(* CODESYS project 3dom.project
   Title: 3dom
   Author: keny
   Version: 0.0.0.14

Project tree, tasks and I/O mapping:
  MyController : TM241CE40T/U, Schneider Electric, order no. TM241CE40T/U, version 4.0.6.18
    application Application
      libraries: Toolbox_Advance, 1.0.1.0 (Schneider Electric); Toolbox, 2.2.0.0 (Schneider Electric)
      task MAST (cyclic, interval 20 ms, priority 15, watchdog 100 ms x 1) calls Program_1
      task VISU_TASK (cyclic, interval 100 ms, priority 30) calls VisuElems.Visu_Prg
      global variables GVL
      visualisation Visualization
      visualisation Visualization_1
    DI : Digital Inputs, Schneider Electric, version 4.0.6.18
        input  M1 : DWORD  // IDW0
        input  lampa_1_kuchania_1_1_wl : BOOL  // IDW0.I0
        input  led_1_kuchnia_1_1_wl : BOOL  // IDW0.I1
        input  kinkiet_1_jadalnia_1_1_wl : BOOL  // IDW0.I2
        input  kinkiet_1_salon_1_1_wl : BOOL  // IDW0.I3
        input  kinkiet_2_salon_1_1_wl : BOOL  // IDW0.I4
        input  kinkiet_3_salon_1_1_wl : BOOL  // IDW0.I5
        input  led_1_salon_1_1_wl : BOOL  // IDW0.I6
        input  lampa_1_salon_1_1_wl : BOOL  // IDW0.I7
        input  lampa_1_jadalnia_1_1_wl : BOOL  // IDW0.I8
        input  kinkiet_1_schody_1_1_wl : BOOL  // IDW0.I9
        input  lampa_zew_wej_1_1_wl : BOOL  // IDW0.I10
        input  lampa_1_przedsionek_1_1_wl : BOOL  // IDW0.I11
        input  lampa_1_korytarz_1_1_wl : BOOL  // IDW0.I12
        input  lampa_1_pokoj_1_1_wl : BOOL  // IDW0.I13
        input  lampa_1_pokoj_2_1_wl : BOOL  // IDW0.I14
        input  kinkiet_1_pokoj_2_1_wl : BOOL  // IDW0.I15
        input  lampa_2_korytarz_1_1_wl : BOOL  // IDW0.I16
        input  lampa_pom_tech_1_1_wl : BOOL  // IDW0.I17
        input  lampa_1_lazienka_1_1_wl : BOOL  // IDW0.I18
        input  kinkiet_1_lazienka_1_1_wl : BOOL  // IDW0.I19
        input  lampa_zew_1_1_wl : BOOL  // IDW0.I20
        input  lampa_zew_2_1_wl : BOOL  // IDW0.I21
        input  lampa_zew_3_1_wl : BOOL  // IDW0.I22
        input  lampa_zew_4_1_wl : BOOL  // IDW0.I23
        input  ibDI_IB1 : BYTE  // IB1
    DQ : Digital Outputs, Schneider Electric, version 4.0.6.18
        output lampa_1_kuchania_1_1_rel : BOOL  // QW0.Q0
        output led_1_kuchnia_1_1_rel : BOOL  // QW0.Q1
        output kinkiet_1_jadalnia_1_1_rel : BOOL  // QW0.Q2
        output kinkiet_1_salon_1_1_rel : BOOL  // QW0.Q3
        output kinkiet_2_salon_1_1_rel : BOOL  // QW0.Q4
        output kinkiet_3_salon_1_1_rel : BOOL  // QW0.Q5
        output led_1_salon_1_1_rel : BOOL  // QW0.Q6
        output lampa_1_salon_1_1_rel : BOOL  // QW0.Q7
        output lampa_1_jadalnia_1_1_rel : BOOL  // QW0.Q8
        output kinkiet_1_schody_1_1_rel : BOOL  // QW0.Q9
        output lampa_zew_wej_1_1_rel : BOOL  // QW0.Q10
        output lampa_1_przedsionek_1_1_rel : BOOL  // QW0.Q11
        output lampa_1_korytarz_1_1_rel : BOOL  // QW0.Q12
        output lampa_1_pokoj_1_1_rel : BOOL  // QW0.Q13
        output lampa_1_pokoj_2_1_rel : BOOL  // QW0.Q14
        output kinkiet_1_pokoj_2_1_rel : BOOL  // QW0.Q15
        unmapped channels: QW0, QB1
    Counters : Counters, Schneider Electric, version 4.0.6.18
    Pulse_Generators : Pulse Generators, Schneider Electric, version 4.0.6.18
    Cartridge_1 : Cartridge, Schneider Electric, version 4.0.6.18
    Cartridge_2 : Cartridge, Schneider Electric, version 4.0.6.18
    IO_Bus : IO bus - TM3, Schneider Electric, version 4.0.6.18
      M2 : TM3DI16/G, Schneider Electric, order no. TM3DI16/G, version 1.0.1.4
          input  M2 : WORD  // IW0
          input  lampa_1_pokoj_3_1_wl : BOOL  // IW0.I0
          input  lampa_1_pom_gosp_1_1_wl : BOOL  // IW0.I1
          input  lampa_1_pokoj_4_1_wl : BOOL  // IW0.I2
          input  lampa_2_pokoj_4_1_wl : BOOL  // IW0.I3
          input  lampa_1_pokoj_5_1_wl : BOOL  // IW0.I4
          input  kinkiet_1_pokoj_5_1_wl : BOOL  // IW0.I5
          input  lampa_1_korytarz_2_1_wl : BOOL  // IW0.I6
          input  led_1_korytarz_2_1_wl : BOOL  // IW0.I7
          input  lampa_1_lazienka_2_1_wl : BOOL  // IW0.I8
          input  kinkiet_1_lazienka_2_1_wl : BOOL  // IW0.I9
          input  kinkiet_2_lazienka_2_1_wl : BOOL  // IW0.I10
          input  lampa_1_pralnia_1_1_wl : BOOL  // IW0.I11
          input  lampa_1_garderoba_1_1_wl : BOOL  // IW0.I12
          input  os_ogrodu_1_1_wl : BOOL  // IW0.I13
          input  kinkiet_4_salon_1_1_wl : BOOL  // IW0.I14
          input  kinkiet_2_schody_1_1_wl : BOOL  // IW0.I15
      M5 : TM3DQ16T/G, Schneider Electric, order no. TM3DQ16T/G, version 1.0.1.4
          output lampa_1_lazienka_2_1_rel : BOOL  // QB0.Q0
          output kinkiet_1_lazienka_2_1_rel : BOOL  // QB0.Q1
          output kinkiet_2_lazienka_2_1_rel : BOOL  // QB0.Q2
          output lampa_1_pralnia_1_1_rel : BOOL  // QB0.Q3
          output lampa_1_garderoba_1_1_rel : BOOL  // QB0.Q4
          output os_ogrodu_1_1_rel : BOOL  // QB0.Q5
          output kinkiet_4_salon_1_1_rel : BOOL  // QB0.Q6
          output kinkiet_2_schody_1_1_rel : BOOL  // QB0.Q7
          output lampa_zew_5_1_rel : BOOL  // QB0.Q8
          unmapped channels: QB0
      M3 : TM3DI16/G, Schneider Electric, order no. TM3DI16/G, version 1.0.1.4
          input  M3 : WORD  // IW0
          input  lampa_zew_5_1_wl : BOOL  // IW0.I0
          input  wlacz_lampy : BOOL  // IW0.I1
          input  wylacz_lampy : BOOL  // IW0.I2
      M4 : TM3DQ16T/G, Schneider Electric, order no. TM3DQ16T/G, version 1.0.1.4
          output lampa_2_korytarz_1_1_rel : BOOL  // QB0.Q0
          output lampa_pom_tech_1_1_rel : BOOL  // QB0.Q1
          output lampa_1_lazienka_1_1_rel : BOOL  // QB0.Q2
          output kinkiet_1_lazienka_1_1_rel : BOOL  // QB0.Q3
          output lampa_zew_1_1_rel : BOOL  // QB0.Q4
          output lampa_zew_2_1_rel : BOOL  // QB0.Q5
          output lampa_zew_3_1_rel : BOOL  // QB0.Q6
          output lampa_zew_4_1_rel : BOOL  // QB0.Q7
          output lampa_1_pokoj_3_1_rel : BOOL  // QB0.Q8
          output lampa_1_pom_gosp_1_1_rel : BOOL  // QB0.Q9
          output lampa_1_pokoj_4_1_rel : BOOL  // QB0.Q10
          output lampa_2_pokoj_4_1_rel : BOOL  // QB0.Q11
          output lampa_1_pokoj_5_1_rel : BOOL  // QB0.Q12
          output kinkiet_1_pokoj_5_1_rel : BOOL  // QB0.Q13
          output lampa_1_korytarz_2_1_rel : BOOL  // QB0.Q14
          output led_1_korytarz_2_1_rel : BOOL  // QB0.Q15
          unmapped channels: QB0
      M6 : TM3DQ16R/G, Schneider Electric, order no. TM3DQ16R/G, version 1.0.1.4
          output zawor_woda_ogrod_1_rel : BOOL  // QW0.Q0
          output ogrzewanie_zawor_1_1_rel : BOOL  // QW0.Q1
          output ogrzewanie_zawor_2_1_rel : BOOL  // QW0.Q2
          output ogrzewanie_zawor_3_1_rel : BOOL  // QW0.Q3
          output ogrzewanie_zawor_4_1_rel : BOOL  // QW0.Q4
          output ogrzewanie_zawor_5_1_rel : BOOL  // QW0.Q5
          output ogrzewanie_zawor_6_1_rel : BOOL  // QW0.Q6
          output ogrzewanie_zawor_7_1_rel : BOOL  // QW0.Q7
          output ogrzewanie_zawor_8_1_rel : BOOL  // QW0.Q8
          unmapped channels: QW0
    COM_Bus : COM bus, Schneider Electric, version 4.0.6.18
    Ethernet_1 : Ethernet Network, Schneider Electric, version 4.0.6.18
        settings: DeviceName = 'nodeZ'; WebServer = TRUE; FTP Server = TRUE; SoMachine Protocol = TRUE; Modbus Server = TRUE; NetManage Protocol = TRUE; SNMP protocol = TRUE; Enable Routing = FALSE; WebVisu protocol = TRUE; DHCP Server Active = TRUE
    Serial_Line_1 : Serial line, Schneider Electric, version 4.0.6.18
      SoMachine_Network_Manager : SoMachine-Network Manager, Schneider Electric, version 4.0.0.2
    Serial_Line_2 : Serial line, Schneider Electric, version 4.0.6.18
      Modbus_Manager : Modbus Manager, Schneider Electric, version 4.0.0.2
  libraries: Standard, * (System)
  function block swichOnOffFUNC [LD]
  function block lightFUNC [LD]
  program Program_1 [LD]
  text list GlobalTextList
  GlobalImagePool
  5ce3da45-db07-42e7-a21c-a00fff4ed8f6|parter.JPG
*)

// MyController/Application/GVL
VAR_GLOBAL 
	;
END_VAR

// Program_1
PROGRAM Program_1
VAR
	lampa_1_kuchania_1_1_DB: swichOnOffFUNC;
	kinkiet_1_jadalnia_1_1_DB: swichOnOffFUNC;
	led_1_kuchnia_1_1_DB: swichOnOffFUNC;
	kinkiet_1_salon_1_1_DB: swichOnOffFUNC;
	kinkiet_2_salon_1_1_DB: swichOnOffFUNC;
	kinkiet_3_salon_1_1_DB: swichOnOffFUNC;
	led_1_salon_1_1_DB: swichOnOffFUNC;
	lampa_1_salon_1_1_DB: swichOnOffFUNC;
	lampa_1_jadalnia_1_1_DB: swichOnOffFUNC;
	kinkiet_1_schody_1_1_DB: swichOnOffFUNC;
	lampa_1_zew_wejsc_1_1_DB: swichOnOffFUNC;
	lampa_1_przedsionek_1_1_DB: swichOnOffFUNC;
	lampa_1_korytarz_1_1_db: swichOnOffFUNC;
	lampa_1_pokoj_1_1_wl_DB: swichOnOffFUNC;
	lampa_1_pokoj_2_1_DB: swichOnOffFUNC;
	kinkiet_1_pokoj_2_1_DB: swichOnOffFUNC;
	lampa_1_korytarz_1_2_DB: swichOnOffFUNC;
	lampa_1_pokoj_1_1_DB: swichOnOffFUNC;
	lampa_2_korytarz_1_1_DB: swichOnOffFUNC;
	lampa_pom_tech_1_1_DB: swichOnOffFUNC;
	lampa_1_laz_1_1_DB: swichOnOffFUNC;
	lampa_1_lazienka_1_1_DB: swichOnOffFUNC;
	kinkiet_1_lazienka_1_1_DB: swichOnOffFUNC;
	lampa_zew_1_1_DB: swichOnOffFUNC;
	lampa_zew_2_1_DB: swichOnOffFUNC;
	lampa_zew_3_1_DB: swichOnOffFUNC;
	lampa_zew_4_1_DB: swichOnOffFUNC;
	lampa_1_pokoj_3_1_DB: swichOnOffFUNC;
	lampa_1_pom_gosp_1_1_DB: swichOnOffFUNC;
	lampa_1_pokoj_4_1_DB: swichOnOffFUNC;
	lampa_2_pokoj_4_1_DB: swichOnOffFUNC;
	lampa_1_pokoj_5_1_DB: swichOnOffFUNC;
	kinkiet_1_pokoj_5_1_DB: swichOnOffFUNC;
	lampa_1_korytarz_2_1_DB: swichOnOffFUNC;
	led_1_korytarz_2_1_DB: swichOnOffFUNC;
	lampa_1_lazienka_2_1_DB: swichOnOffFUNC;
	kinkiet_1_lazienka_2_1_DB: swichOnOffFUNC;
	kinkiet_2_lazienka_2_1_DB: swichOnOffFUNC;
	lampa_1_pralnia_1_1_DB: swichOnOffFUNC;
	lampa_1_garderoba_1_1_DB: swichOnOffFUNC;
	os_ogrodu_1_1_DB: swichOnOffFUNC;
	kinkiet_4_salon_1_1_DB: swichOnOffFUNC;
	kinkiet_2_schody_1_1_DB: swichOnOffFUNC;
	lampa_zew_5_1_DB: swichOnOffFUNC;
	wlacz_lampy_DB: swichOnOffFUNC;
	lamp_zewnetrzna_1: BOOL;
	lampa_zewnetrzna_5_visu: BOOL;
	lampa_1_kuchania_visu: BOOL;
	led_1_kuchnia_1_1_visu: BOOL;
	kinkiet_1_jadalnia_1_1_visu: BOOL;
	kinkiet_1_salon_1_1_visu: BOOL;
	kinkiet_2_salon_1_1_visu: BOOL;
	kinkiet_3_salon_1_1_visu: BOOL;
	lampa_1_salon_1_1_visu: BOOL;
	lampa_1_jadalnia_1_1_visu: BOOL;
	kinkiet_1_schody_1_1_visu: BOOL;
	lampa_zew_wej_1_1_visu: BOOL;
	lampa_1_przedsionek_1_1_visu: BOOL;
	lampa_1_korytarz_1_1_visu: BOOL;
	lampa_1_pokoj_1_1_visu: BOOL;
	lampa_1_pokoj_2_1_visu: BOOL;
	led_1_kuchnia_visu: BOOL;
	lampa_2_korytarz_1_1_VISU: BOOL;
	kinkiet_1_pokoj_2_1_visu: BOOL;
	lampa_pom_tech_1_1_visu: BOOL;
	lampa_1_lazienka_1_1_visu: BOOL;
	kinkiet_1_lazienka_1_1_visu: BOOL;
	lampa_zew_1_1_visu: BOOL;
	lampa_zew_2_1_visu: BOOL;
	lampa_zew_3_1_visu: BOOL;
	lampa_zew_4_1_visu: BOOL;
	lampa_1_pokoj_3_1_visu: BOOL;
	lampa_1_pom_gosp_1_1_visu: BOOL;
	lampa_1_pokoj_4_1_visu: BOOL;
	lampa_2_pokoj_4_1_visu: BOOL;
	lampa_1_pokoj_5_1_visu: BOOL;
	kinkiet_1_pokoj_5_1_visu: BOOL;
	lampa_1_korytarz_2_1_visu: BOOL;
	led_1_korytarz_2_1_visu: BOOL;
	lampa_1_lazienka_2_1_visu: BOOL;
	kinkiet_1_lazienka_2_1_visu: BOOL;
	kinkiet_2_lazienka_2_1_visu: BOOL;
	lampa_1_pralnia_1_1_visu: BOOL;
	lampa_1_garderoba_1_1_visu: BOOL;
	os_ogrodu_1_1_visu: BOOL;
	kinkiet_4_salon_1_1_visu: BOOL;
	kinkiet_2_schody_1_1_visu: BOOL;
	lampa_zew_5_1_visu: BOOL;
	led_1_salon_1_1_visu: BOOL;
END_VAR

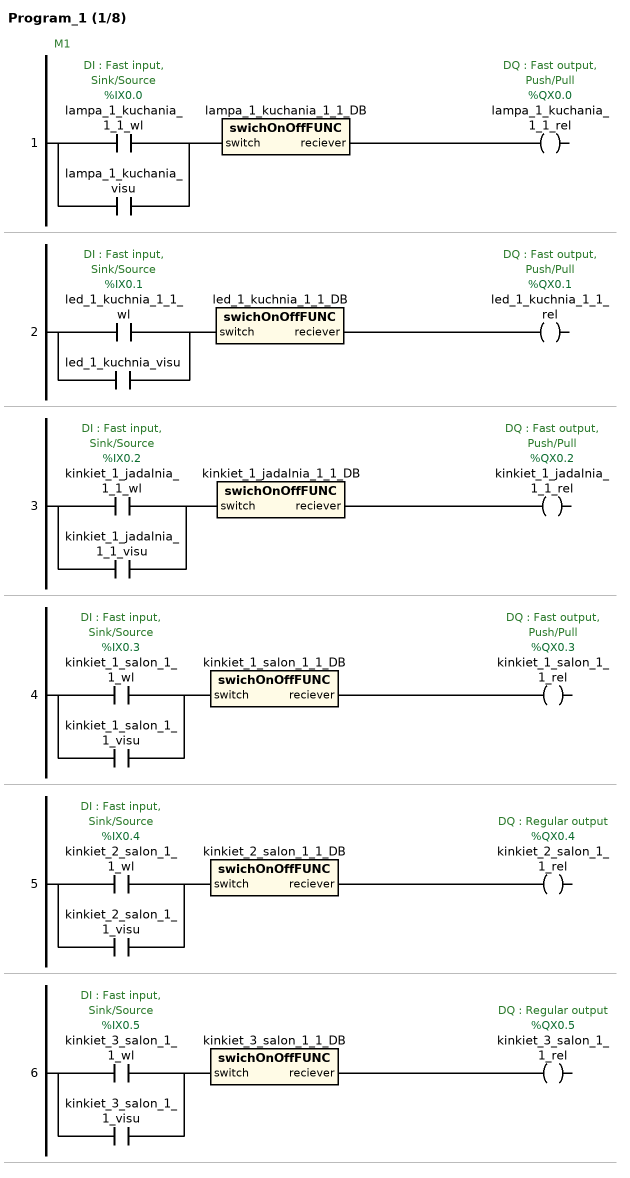
// NETWORK 1
// M1
//   lampa_1_kuchania_1_1_wl: DI : Fast input, Sink/Source | AT %IX0.0
//   lampa_1_kuchania_1_1_rel: DQ : Fast output, Push/Pull | AT %QX0.0
lampa_1_kuchania_1_1_DB(switch := lampa_1_kuchania_1_1_wl OR lampa_1_kuchania_visu); // swichOnOffFUNC
lampa_1_kuchania_1_1_rel := lampa_1_kuchania_1_1_DB.reciever;

// NETWORK 2
//   led_1_kuchnia_1_1_wl: DI : Fast input, Sink/Source | AT %IX0.1
//   led_1_kuchnia_1_1_rel: DQ : Fast output, Push/Pull | AT %QX0.1
led_1_kuchnia_1_1_DB(switch := led_1_kuchnia_1_1_wl OR led_1_kuchnia_visu); // swichOnOffFUNC
led_1_kuchnia_1_1_rel := led_1_kuchnia_1_1_DB.reciever;

// NETWORK 3
//   kinkiet_1_jadalnia_1_1_wl: DI : Fast input, Sink/Source | AT %IX0.2
//   kinkiet_1_jadalnia_1_1_rel: DQ : Fast output, Push/Pull | AT %QX0.2
kinkiet_1_jadalnia_1_1_DB(switch := kinkiet_1_jadalnia_1_1_wl OR kinkiet_1_jadalnia_1_1_visu); // swichOnOffFUNC
kinkiet_1_jadalnia_1_1_rel := kinkiet_1_jadalnia_1_1_DB.reciever;

// NETWORK 4
//   kinkiet_1_salon_1_1_wl: DI : Fast input, Sink/Source | AT %IX0.3
//   kinkiet_1_salon_1_1_rel: DQ : Fast output, Push/Pull | AT %QX0.3
kinkiet_1_salon_1_1_DB(switch := kinkiet_1_salon_1_1_wl OR kinkiet_1_salon_1_1_visu); // swichOnOffFUNC
kinkiet_1_salon_1_1_rel := kinkiet_1_salon_1_1_DB.reciever;

// NETWORK 5
//   kinkiet_2_salon_1_1_wl: DI : Fast input, Sink/Source | AT %IX0.4
//   kinkiet_2_salon_1_1_rel: DQ : Regular output | AT %QX0.4
kinkiet_2_salon_1_1_DB(switch := kinkiet_2_salon_1_1_wl OR kinkiet_2_salon_1_1_visu); // swichOnOffFUNC
kinkiet_2_salon_1_1_rel := kinkiet_2_salon_1_1_DB.reciever;

// NETWORK 6
//   kinkiet_3_salon_1_1_wl: DI : Fast input, Sink/Source | AT %IX0.5
//   kinkiet_3_salon_1_1_rel: DQ : Regular output | AT %QX0.5
kinkiet_3_salon_1_1_DB(switch := kinkiet_3_salon_1_1_wl OR kinkiet_3_salon_1_1_visu); // swichOnOffFUNC
kinkiet_3_salon_1_1_rel := kinkiet_3_salon_1_1_DB.reciever;

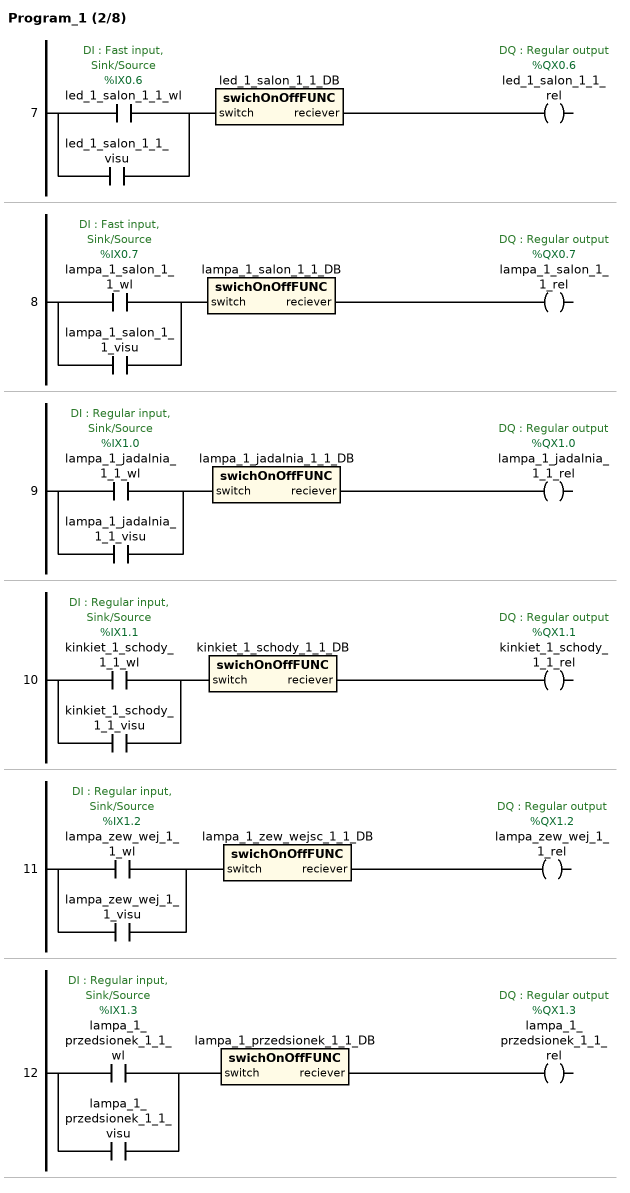
// NETWORK 7
//   led_1_salon_1_1_wl: DI : Fast input, Sink/Source | AT %IX0.6
//   led_1_salon_1_1_rel: DQ : Regular output | AT %QX0.6
led_1_salon_1_1_DB(switch := led_1_salon_1_1_wl OR led_1_salon_1_1_visu); // swichOnOffFUNC
led_1_salon_1_1_rel := led_1_salon_1_1_DB.reciever;

// NETWORK 8
//   lampa_1_salon_1_1_wl: DI : Fast input, Sink/Source | AT %IX0.7
//   lampa_1_salon_1_1_rel: DQ : Regular output | AT %QX0.7
lampa_1_salon_1_1_DB(switch := lampa_1_salon_1_1_wl OR lampa_1_salon_1_1_visu); // swichOnOffFUNC
lampa_1_salon_1_1_rel := lampa_1_salon_1_1_DB.reciever;

// NETWORK 9
//   lampa_1_jadalnia_1_1_wl: DI : Regular input, Sink/Source | AT %IX1.0
//   lampa_1_jadalnia_1_1_rel: DQ : Regular output | AT %QX1.0
lampa_1_jadalnia_1_1_DB(switch := lampa_1_jadalnia_1_1_wl OR lampa_1_jadalnia_1_1_visu); // swichOnOffFUNC
lampa_1_jadalnia_1_1_rel := lampa_1_jadalnia_1_1_DB.reciever;

// NETWORK 10
//   kinkiet_1_schody_1_1_wl: DI : Regular input, Sink/Source | AT %IX1.1
//   kinkiet_1_schody_1_1_rel: DQ : Regular output | AT %QX1.1
kinkiet_1_schody_1_1_DB(switch := kinkiet_1_schody_1_1_wl OR kinkiet_1_schody_1_1_visu); // swichOnOffFUNC
kinkiet_1_schody_1_1_rel := kinkiet_1_schody_1_1_DB.reciever;

// NETWORK 11
//   lampa_zew_wej_1_1_wl: DI : Regular input, Sink/Source | AT %IX1.2
//   lampa_zew_wej_1_1_rel: DQ : Regular output | AT %QX1.2
lampa_1_zew_wejsc_1_1_DB(switch := lampa_zew_wej_1_1_wl OR lampa_zew_wej_1_1_visu); // swichOnOffFUNC
lampa_zew_wej_1_1_rel := lampa_1_zew_wejsc_1_1_DB.reciever;

// NETWORK 12
//   lampa_1_przedsionek_1_1_wl: DI : Regular input, Sink/Source | AT %IX1.3
//   lampa_1_przedsionek_1_1_rel: DQ : Regular output | AT %QX1.3
lampa_1_przedsionek_1_1_DB(switch := lampa_1_przedsionek_1_1_wl OR lampa_1_przedsionek_1_1_visu); // swichOnOffFUNC
lampa_1_przedsionek_1_1_rel := lampa_1_przedsionek_1_1_DB.reciever;

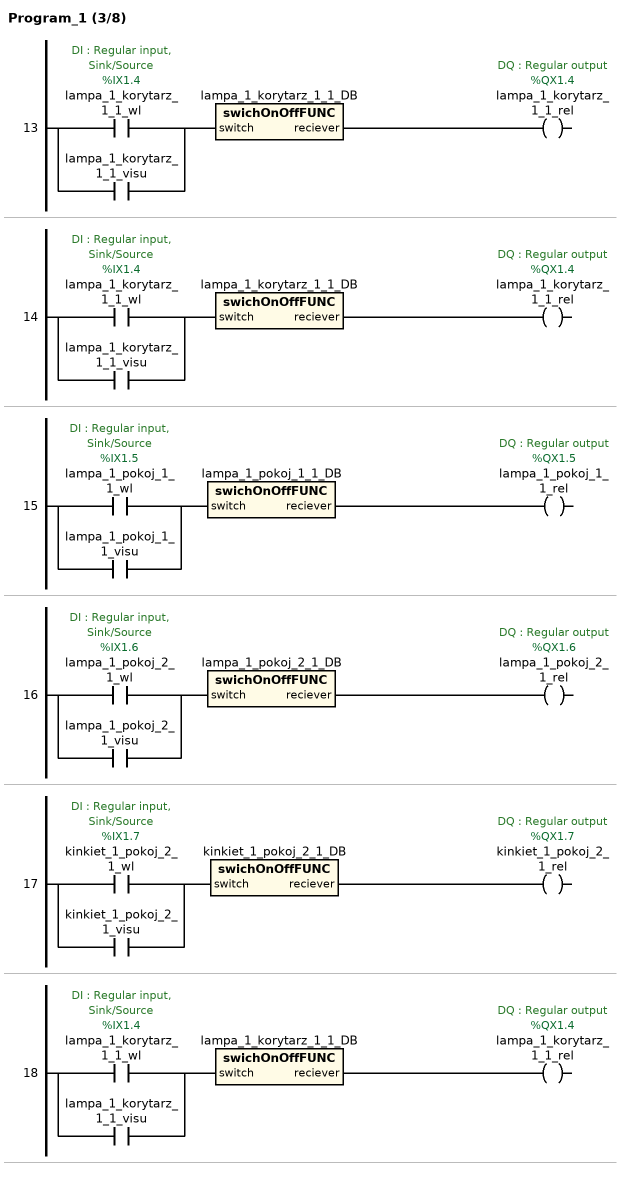
// NETWORK 13
//   lampa_1_korytarz_1_1_wl: DI : Regular input, Sink/Source | AT %IX1.4
//   lampa_1_korytarz_1_1_rel: DQ : Regular output | AT %QX1.4
lampa_1_korytarz_1_1_DB(switch := lampa_1_korytarz_1_1_wl OR lampa_1_korytarz_1_1_visu); // swichOnOffFUNC
lampa_1_korytarz_1_1_rel := lampa_1_korytarz_1_1_DB.reciever;

// NETWORK 14
//   lampa_1_korytarz_1_1_wl: DI : Regular input, Sink/Source | AT %IX1.4
//   lampa_1_korytarz_1_1_rel: DQ : Regular output | AT %QX1.4
lampa_1_korytarz_1_1_DB(switch := lampa_1_korytarz_1_1_wl OR lampa_1_korytarz_1_1_visu); // swichOnOffFUNC
lampa_1_korytarz_1_1_rel := lampa_1_korytarz_1_1_DB.reciever;

// NETWORK 15
//   lampa_1_pokoj_1_1_wl: DI : Regular input, Sink/Source | AT %IX1.5
//   lampa_1_pokoj_1_1_rel: DQ : Regular output | AT %QX1.5
lampa_1_pokoj_1_1_DB(switch := lampa_1_pokoj_1_1_wl OR lampa_1_pokoj_1_1_visu); // swichOnOffFUNC
lampa_1_pokoj_1_1_rel := lampa_1_pokoj_1_1_DB.reciever;

// NETWORK 16
//   lampa_1_pokoj_2_1_wl: DI : Regular input, Sink/Source | AT %IX1.6
//   lampa_1_pokoj_2_1_rel: DQ : Regular output | AT %QX1.6
lampa_1_pokoj_2_1_DB(switch := lampa_1_pokoj_2_1_wl OR lampa_1_pokoj_2_1_visu); // swichOnOffFUNC
lampa_1_pokoj_2_1_rel := lampa_1_pokoj_2_1_DB.reciever;

// NETWORK 17
//   kinkiet_1_pokoj_2_1_wl: DI : Regular input, Sink/Source | AT %IX1.7
//   kinkiet_1_pokoj_2_1_rel: DQ : Regular output | AT %QX1.7
kinkiet_1_pokoj_2_1_DB(switch := kinkiet_1_pokoj_2_1_wl OR kinkiet_1_pokoj_2_1_visu); // swichOnOffFUNC
kinkiet_1_pokoj_2_1_rel := kinkiet_1_pokoj_2_1_DB.reciever;

// NETWORK 18
//   lampa_1_korytarz_1_1_wl: DI : Regular input, Sink/Source | AT %IX1.4
//   lampa_1_korytarz_1_1_rel: DQ : Regular output | AT %QX1.4
lampa_1_korytarz_1_1_DB(switch := lampa_1_korytarz_1_1_wl OR lampa_1_korytarz_1_1_visu); // swichOnOffFUNC
lampa_1_korytarz_1_1_rel := lampa_1_korytarz_1_1_DB.reciever;

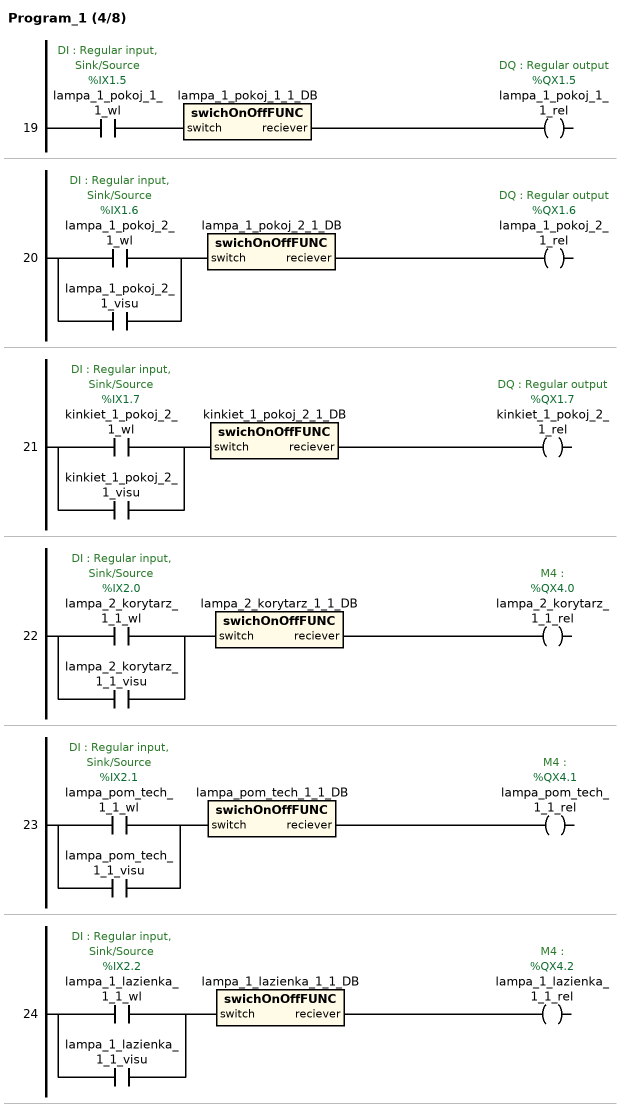
// NETWORK 19
//   lampa_1_pokoj_1_1_wl: DI : Regular input, Sink/Source | AT %IX1.5
//   lampa_1_pokoj_1_1_rel: DQ : Regular output | AT %QX1.5
lampa_1_pokoj_1_1_DB(switch := lampa_1_pokoj_1_1_wl); // swichOnOffFUNC
lampa_1_pokoj_1_1_rel := lampa_1_pokoj_1_1_DB.reciever;

// NETWORK 20
//   lampa_1_pokoj_2_1_wl: DI : Regular input, Sink/Source | AT %IX1.6
//   lampa_1_pokoj_2_1_rel: DQ : Regular output | AT %QX1.6
lampa_1_pokoj_2_1_DB(switch := lampa_1_pokoj_2_1_wl OR lampa_1_pokoj_2_1_visu); // swichOnOffFUNC
lampa_1_pokoj_2_1_rel := lampa_1_pokoj_2_1_DB.reciever;

// NETWORK 21
//   kinkiet_1_pokoj_2_1_wl: DI : Regular input, Sink/Source | AT %IX1.7
//   kinkiet_1_pokoj_2_1_rel: DQ : Regular output | AT %QX1.7
kinkiet_1_pokoj_2_1_DB(switch := kinkiet_1_pokoj_2_1_wl OR kinkiet_1_pokoj_2_1_visu); // swichOnOffFUNC
kinkiet_1_pokoj_2_1_rel := kinkiet_1_pokoj_2_1_DB.reciever;

// NETWORK 22
//   lampa_2_korytarz_1_1_wl: DI : Regular input, Sink/Source | AT %IX2.0
//   lampa_2_korytarz_1_1_rel: M4 : | AT %QX4.0
lampa_2_korytarz_1_1_DB(switch := lampa_2_korytarz_1_1_wl OR lampa_2_korytarz_1_1_visu); // swichOnOffFUNC
lampa_2_korytarz_1_1_rel := lampa_2_korytarz_1_1_DB.reciever;

// NETWORK 23
//   lampa_pom_tech_1_1_wl: DI : Regular input, Sink/Source | AT %IX2.1
//   lampa_pom_tech_1_1_rel: M4 : | AT %QX4.1
lampa_pom_tech_1_1_DB(switch := lampa_pom_tech_1_1_wl OR lampa_pom_tech_1_1_visu); // swichOnOffFUNC
lampa_pom_tech_1_1_rel := lampa_pom_tech_1_1_DB.reciever;

// NETWORK 24
//   lampa_1_lazienka_1_1_wl: DI : Regular input, Sink/Source | AT %IX2.2
//   lampa_1_lazienka_1_1_rel: M4 : | AT %QX4.2
lampa_1_lazienka_1_1_DB(switch := lampa_1_lazienka_1_1_wl OR lampa_1_lazienka_1_1_visu); // swichOnOffFUNC
lampa_1_lazienka_1_1_rel := lampa_1_lazienka_1_1_DB.reciever;

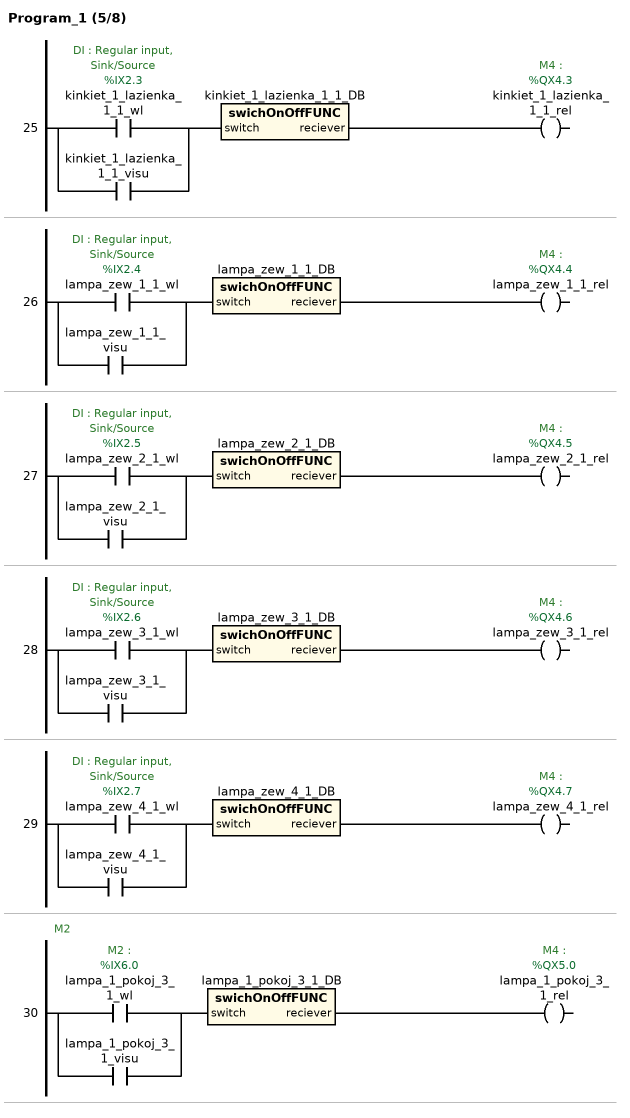
// NETWORK 25
//   kinkiet_1_lazienka_1_1_wl: DI : Regular input, Sink/Source | AT %IX2.3
//   kinkiet_1_lazienka_1_1_rel: M4 : | AT %QX4.3
kinkiet_1_lazienka_1_1_DB(switch := kinkiet_1_lazienka_1_1_wl OR kinkiet_1_lazienka_1_1_visu); // swichOnOffFUNC
kinkiet_1_lazienka_1_1_rel := kinkiet_1_lazienka_1_1_DB.reciever;

// NETWORK 26
//   lampa_zew_1_1_wl: DI : Regular input, Sink/Source | AT %IX2.4
//   lampa_zew_1_1_rel: M4 : | AT %QX4.4
lampa_zew_1_1_DB(switch := lampa_zew_1_1_wl OR lampa_zew_1_1_visu); // swichOnOffFUNC
lampa_zew_1_1_rel := lampa_zew_1_1_DB.reciever;

// NETWORK 27
//   lampa_zew_2_1_wl: DI : Regular input, Sink/Source | AT %IX2.5
//   lampa_zew_2_1_rel: M4 : | AT %QX4.5
lampa_zew_2_1_DB(switch := lampa_zew_2_1_wl OR lampa_zew_2_1_visu); // swichOnOffFUNC
lampa_zew_2_1_rel := lampa_zew_2_1_DB.reciever;

// NETWORK 28
//   lampa_zew_3_1_wl: DI : Regular input, Sink/Source | AT %IX2.6
//   lampa_zew_3_1_rel: M4 : | AT %QX4.6
lampa_zew_3_1_DB(switch := lampa_zew_3_1_wl OR lampa_zew_3_1_visu); // swichOnOffFUNC
lampa_zew_3_1_rel := lampa_zew_3_1_DB.reciever;

// NETWORK 29
//   lampa_zew_4_1_wl: DI : Regular input, Sink/Source | AT %IX2.7
//   lampa_zew_4_1_rel: M4 : | AT %QX4.7
lampa_zew_4_1_DB(switch := lampa_zew_4_1_wl OR lampa_zew_4_1_visu); // swichOnOffFUNC
lampa_zew_4_1_rel := lampa_zew_4_1_DB.reciever;

// NETWORK 30
// M2
//   lampa_1_pokoj_3_1_wl: M2 : | AT %IX6.0
//   lampa_1_pokoj_3_1_rel: M4 : | AT %QX5.0
lampa_1_pokoj_3_1_DB(switch := lampa_1_pokoj_3_1_wl OR lampa_1_pokoj_3_1_visu); // swichOnOffFUNC
lampa_1_pokoj_3_1_rel := lampa_1_pokoj_3_1_DB.reciever;

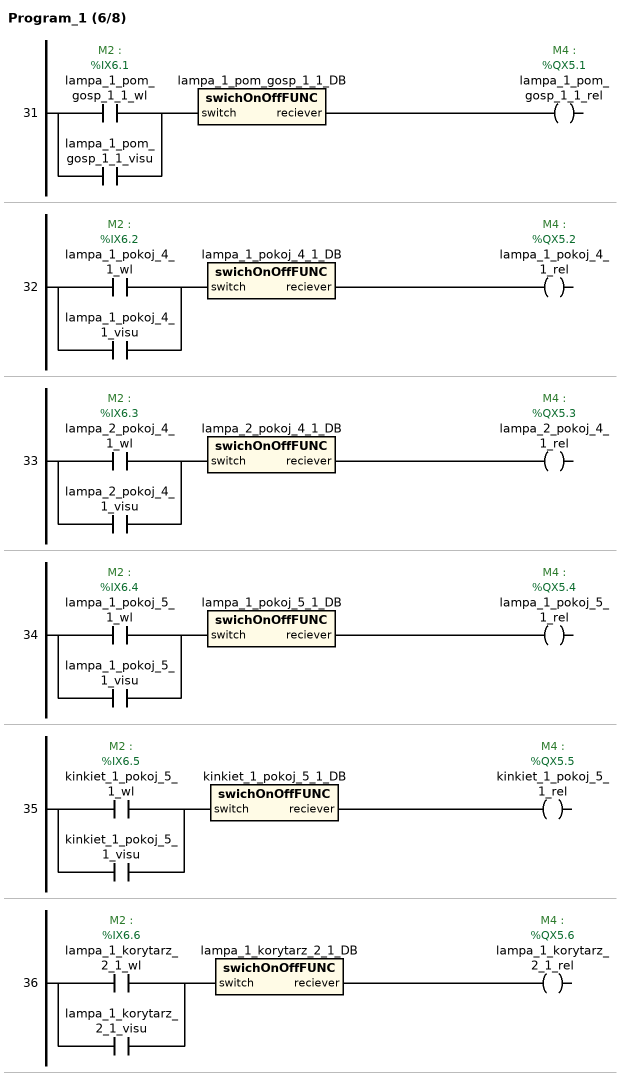
// NETWORK 31
//   lampa_1_pom_gosp_1_1_wl: M2 : | AT %IX6.1
//   lampa_1_pom_gosp_1_1_rel: M4 : | AT %QX5.1
lampa_1_pom_gosp_1_1_DB(switch := lampa_1_pom_gosp_1_1_wl OR lampa_1_pom_gosp_1_1_visu); // swichOnOffFUNC
lampa_1_pom_gosp_1_1_rel := lampa_1_pom_gosp_1_1_DB.reciever;

// NETWORK 32
//   lampa_1_pokoj_4_1_wl: M2 : | AT %IX6.2
//   lampa_1_pokoj_4_1_rel: M4 : | AT %QX5.2
lampa_1_pokoj_4_1_DB(switch := lampa_1_pokoj_4_1_wl OR lampa_1_pokoj_4_1_visu); // swichOnOffFUNC
lampa_1_pokoj_4_1_rel := lampa_1_pokoj_4_1_DB.reciever;

// NETWORK 33
//   lampa_2_pokoj_4_1_wl: M2 : | AT %IX6.3
//   lampa_2_pokoj_4_1_rel: M4 : | AT %QX5.3
lampa_2_pokoj_4_1_DB(switch := lampa_2_pokoj_4_1_wl OR lampa_2_pokoj_4_1_visu); // swichOnOffFUNC
lampa_2_pokoj_4_1_rel := lampa_2_pokoj_4_1_DB.reciever;

// NETWORK 34
//   lampa_1_pokoj_5_1_wl: M2 : | AT %IX6.4
//   lampa_1_pokoj_5_1_rel: M4 : | AT %QX5.4
lampa_1_pokoj_5_1_DB(switch := lampa_1_pokoj_5_1_wl OR lampa_1_pokoj_5_1_visu); // swichOnOffFUNC
lampa_1_pokoj_5_1_rel := lampa_1_pokoj_5_1_DB.reciever;

// NETWORK 35
//   kinkiet_1_pokoj_5_1_wl: M2 : | AT %IX6.5
//   kinkiet_1_pokoj_5_1_rel: M4 : | AT %QX5.5
kinkiet_1_pokoj_5_1_DB(switch := kinkiet_1_pokoj_5_1_wl OR kinkiet_1_pokoj_5_1_visu); // swichOnOffFUNC
kinkiet_1_pokoj_5_1_rel := kinkiet_1_pokoj_5_1_DB.reciever;

// NETWORK 36
//   lampa_1_korytarz_2_1_wl: M2 : | AT %IX6.6
//   lampa_1_korytarz_2_1_rel: M4 : | AT %QX5.6
lampa_1_korytarz_2_1_DB(switch := lampa_1_korytarz_2_1_wl OR lampa_1_korytarz_2_1_visu); // swichOnOffFUNC
lampa_1_korytarz_2_1_rel := lampa_1_korytarz_2_1_DB.reciever;

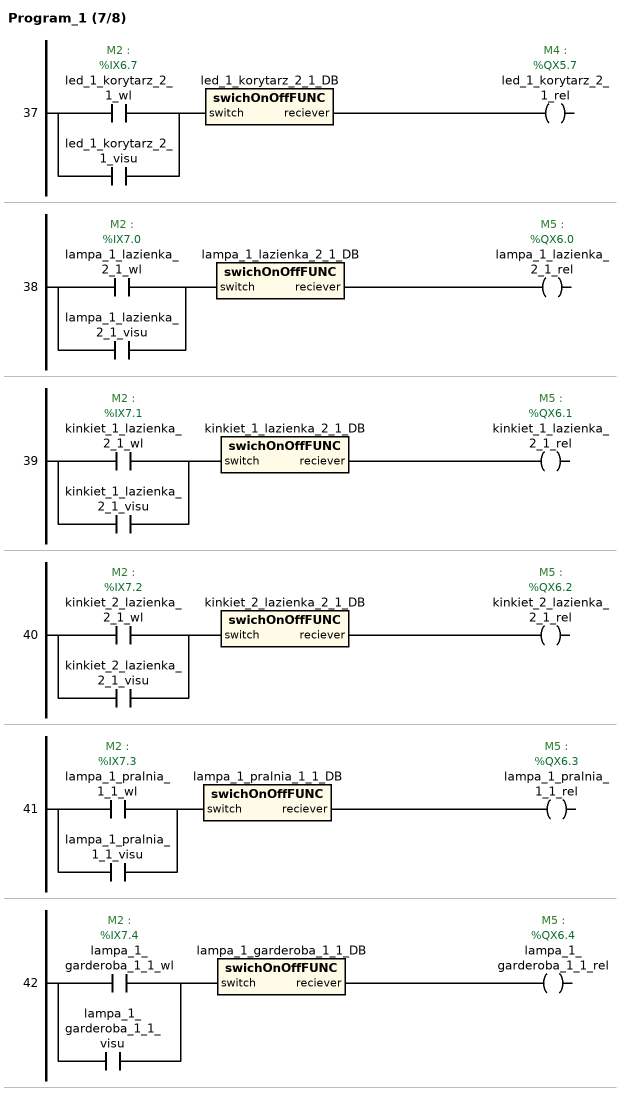
// NETWORK 37
//   led_1_korytarz_2_1_wl: M2 : | AT %IX6.7
//   led_1_korytarz_2_1_rel: M4 : | AT %QX5.7
led_1_korytarz_2_1_DB(switch := led_1_korytarz_2_1_wl OR led_1_korytarz_2_1_visu); // swichOnOffFUNC
led_1_korytarz_2_1_rel := led_1_korytarz_2_1_DB.reciever;

// NETWORK 38
//   lampa_1_lazienka_2_1_wl: M2 : | AT %IX7.0
//   lampa_1_lazienka_2_1_rel: M5 : | AT %QX6.0
lampa_1_lazienka_2_1_DB(switch := lampa_1_lazienka_2_1_wl OR lampa_1_lazienka_2_1_visu); // swichOnOffFUNC
lampa_1_lazienka_2_1_rel := lampa_1_lazienka_2_1_DB.reciever;

// NETWORK 39
//   kinkiet_1_lazienka_2_1_wl: M2 : | AT %IX7.1
//   kinkiet_1_lazienka_2_1_rel: M5 : | AT %QX6.1
kinkiet_1_lazienka_2_1_DB(switch := kinkiet_1_lazienka_2_1_wl OR kinkiet_1_lazienka_2_1_visu); // swichOnOffFUNC
kinkiet_1_lazienka_2_1_rel := kinkiet_1_lazienka_2_1_DB.reciever;

// NETWORK 40
//   kinkiet_2_lazienka_2_1_wl: M2 : | AT %IX7.2
//   kinkiet_2_lazienka_2_1_rel: M5 : | AT %QX6.2
kinkiet_2_lazienka_2_1_DB(switch := kinkiet_2_lazienka_2_1_wl OR kinkiet_2_lazienka_2_1_visu); // swichOnOffFUNC
kinkiet_2_lazienka_2_1_rel := kinkiet_2_lazienka_2_1_DB.reciever;

// NETWORK 41
//   lampa_1_pralnia_1_1_wl: M2 : | AT %IX7.3
//   lampa_1_pralnia_1_1_rel: M5 : | AT %QX6.3
lampa_1_pralnia_1_1_DB(switch := lampa_1_pralnia_1_1_wl OR lampa_1_pralnia_1_1_visu); // swichOnOffFUNC
lampa_1_pralnia_1_1_rel := lampa_1_pralnia_1_1_DB.reciever;

// NETWORK 42
//   lampa_1_garderoba_1_1_wl: M2 : | AT %IX7.4
//   lampa_1_garderoba_1_1_rel: M5 : | AT %QX6.4
lampa_1_garderoba_1_1_DB(switch := lampa_1_garderoba_1_1_wl OR lampa_1_garderoba_1_1_visu); // swichOnOffFUNC
lampa_1_garderoba_1_1_rel := lampa_1_garderoba_1_1_DB.reciever;

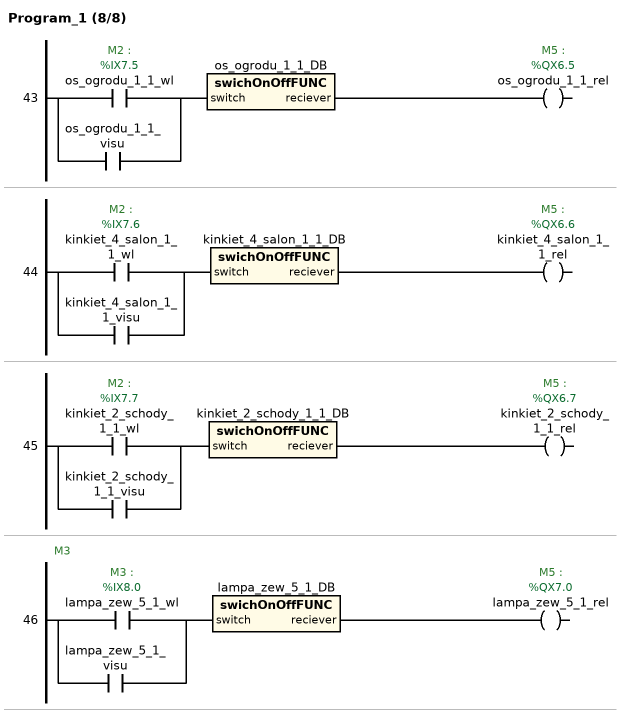
// NETWORK 43
//   os_ogrodu_1_1_wl: M2 : | AT %IX7.5
//   os_ogrodu_1_1_rel: M5 : | AT %QX6.5
os_ogrodu_1_1_DB(switch := os_ogrodu_1_1_wl OR os_ogrodu_1_1_visu); // swichOnOffFUNC
os_ogrodu_1_1_rel := os_ogrodu_1_1_DB.reciever;

// NETWORK 44
//   kinkiet_4_salon_1_1_wl: M2 : | AT %IX7.6
//   kinkiet_4_salon_1_1_rel: M5 : | AT %QX6.6
kinkiet_4_salon_1_1_DB(switch := kinkiet_4_salon_1_1_wl OR kinkiet_4_salon_1_1_visu); // swichOnOffFUNC
kinkiet_4_salon_1_1_rel := kinkiet_4_salon_1_1_DB.reciever;

// NETWORK 45
//   kinkiet_2_schody_1_1_wl: M2 : | AT %IX7.7
//   kinkiet_2_schody_1_1_rel: M5 : | AT %QX6.7
kinkiet_2_schody_1_1_DB(switch := kinkiet_2_schody_1_1_wl OR kinkiet_2_schody_1_1_visu); // swichOnOffFUNC
kinkiet_2_schody_1_1_rel := kinkiet_2_schody_1_1_DB.reciever;

// NETWORK 46
// M3
//   lampa_zew_5_1_wl: M3 : | AT %IX8.0
//   lampa_zew_5_1_rel: M5 : | AT %QX7.0
lampa_zew_5_1_DB(switch := lampa_zew_5_1_wl OR lampa_zew_5_1_visu); // swichOnOffFUNC
lampa_zew_5_1_rel := lampa_zew_5_1_DB.reciever;

END_PROGRAM

// swichOnOffFUNC
FUNCTION_BLOCK PUBLIC swichOnOffFUNC
VAR_INPUT
	switch: BOOL;
END_VAR
VAR_OUTPUT
	reciever: BOOL;
END_VAR
VAR
	changed: BOOL;
	switch_ON: BOOL;
END_VAR
VAR // added by the converter: edge detectors and wires of the graphical bodies
    _rt1 : R_TRIG;
    _w1, _w2 : BOOL;
END_VAR

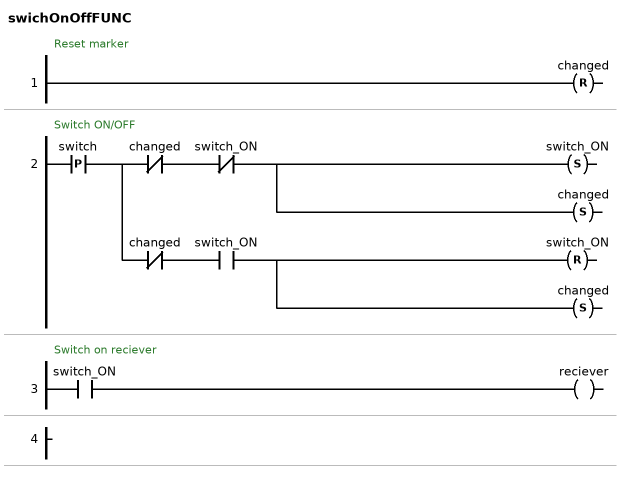
// NETWORK 1
// Reset marker
changed R= TRUE;

// NETWORK 2
// Switch ON/OFF
_rt1(CLK := switch);
_w1 := _rt1.Q AND NOT changed AND NOT switch_ON;
switch_ON S= _w1;
changed S= _w1;
_w2 := _rt1.Q AND NOT changed AND switch_ON;
switch_ON R= _w2;
changed S= _w2;

// NETWORK 3
// Switch on reciever
reciever := switch_ON;

// NETWORK 4

END_FUNCTION_BLOCK

// lightFUNC
FUNCTION_BLOCK PUBLIC lightFUNC
VAR_INPUT
	light_switch: BOOL;
END_VAR
VAR_OUTPUT
	light_bulb: BOOL;
END_VAR
VAR
	changed: BOOL;
	light_ON: BOOL;
END_VAR
VAR // added by the converter: edge detectors and wires of the graphical bodies
    _rt1 : R_TRIG;
    _w1, _w2 : BOOL;
END_VAR

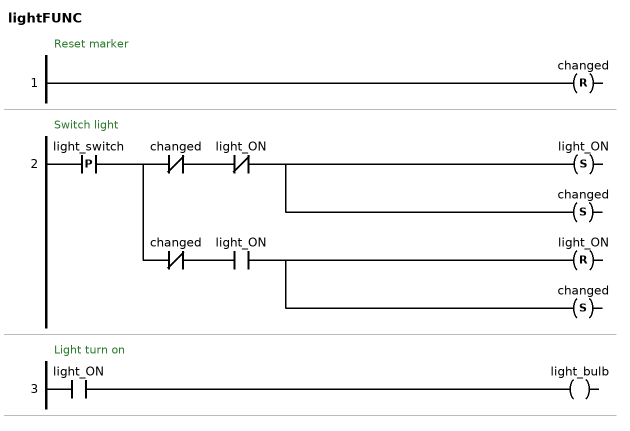
// NETWORK 1
// Reset marker
changed R= TRUE;

// NETWORK 2
// Switch light
_rt1(CLK := light_switch);
_w1 := _rt1.Q AND NOT changed AND NOT light_ON;
light_ON S= _w1;
changed S= _w1;
_w2 := _rt1.Q AND NOT changed AND light_ON;
light_ON R= _w2;
changed S= _w2;

// NETWORK 3
// Light turn on
light_bulb := light_ON;

END_FUNCTION_BLOCK

// MyController/Application/Visualization
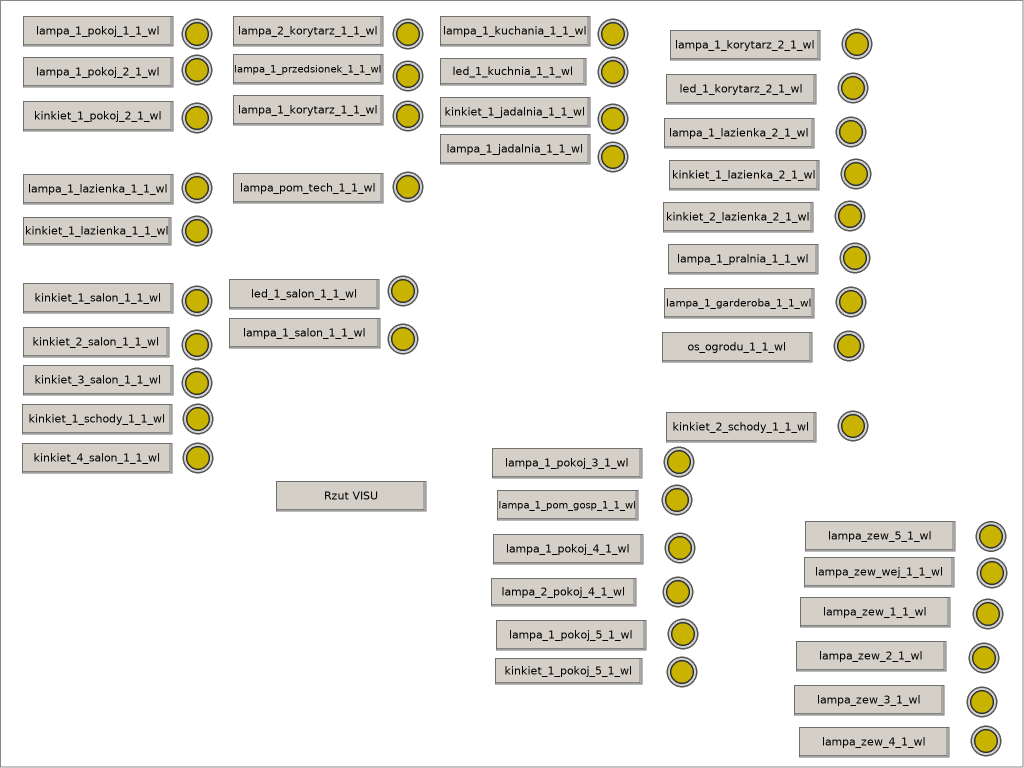
VISUALIZATION Visualization  // 1024x768
    Button (440,16 150x30), "lampa_1_kuchania_1_1_wl"
        tap Program_1.lampa_1_kuchania_visu
    Lamp1 (595,16 36x36), variable: lampa_1_kuchania_1_1_rel, style: Lamp-Lamp1-Yellow
    Button (440,58 146x27), "led_1_kuchnia_1_1_wl"
        tap Program_1.led_1_kuchnia_visu
    Lamp1 (595,54 36x36), variable: led_1_kuchnia_1_1_rel, style: Lamp-Lamp1-Yellow
    Button (440,97 150x30), "kinkiet_1_jadalnia_1_1_wl"
        tap Program_1.kinkiet_1_jadalnia_1_1_visu
    Lamp1 (595,101 36x36), variable: kinkiet_1_jadalnia_1_1_rel, style: Lamp-Lamp1-Yellow
    Button (23,283 150x30), "kinkiet_1_salon_1_1_wl"
        tap Program_1.kinkiet_1_salon_1_1_visu
    Lamp1 (179,283 36x36), variable: kinkiet_1_salon_1_1_rel, style: Lamp-Lamp1-Yellow
    Button (23,327 146x30), "kinkiet_2_salon_1_1_wl"
        tap Program_1.kinkiet_2_salon_1_1_visu
    Lamp1 (179,327 36x36), variable: kinkiet_2_salon_1_1_rel, style: Lamp-Lamp1-Yellow
    Button (23,365 150x30), "kinkiet_3_salon_1_1_wl"
        tap Program_1.kinkiet_3_salon_1_1_visu
    Lamp1 (179,365 36x36), variable: kinkiet_3_salon_1_1_rel, style: Lamp-Lamp1-Yellow
    Button (229,279 150x30), "led_1_salon_1_1_wl"
        tap Program_1.led_1_salon_1_1_visu
    Lamp1 (385,273 36x36), variable: led_1_salon_1_1_rel, style: Lamp-Lamp1-Yellow
    Button (229,318 151x30), "lampa_1_salon_1_1_wl"
        tap Program_1.lampa_1_salon_1_1_visu
    Lamp1 (385,321 36x36), variable: lampa_1_salon_1_1_rel, style: Lamp-Lamp1-Yellow
    Button (440,134 150x30), "lampa_1_jadalnia_1_1_wl"
        tap Program_1.lampa_1_jadalnia_1_1_visu
    Lamp1 (595,139 36x36), variable: lampa_1_jadalnia_1_1_rel, style: Lamp-Lamp1-Yellow
    Button (22,404 150x30), "kinkiet_1_schody_1_1_wl"
        tap Program_1.kinkiet_1_schody_1_1_visu
    Lamp1 (180,401 36x36), variable: kinkiet_1_schody_1_1_rel, style: Lamp-Lamp1-Yellow
    Button (804,557 150x30), "lampa_zew_wej_1_1_wl"
        tap Program_1.lampa_zew_wej_1_1_visu
    Lamp1 (974,555 36x36), variable: lampa_zew_wej_1_1_rel, style: Lamp-Lamp1-Yellow
    Button (233,54 150x30), "lampa_1_przedsionek_1_1_wl"
        tap Program_1.lampa_1_przedsionek_1_1_visu
    Lamp1 (390,58 36x36), variable: lampa_1_przedsionek_1_1_rel, style: Lamp-Lamp1-Yellow
    Button (233,95 150x30), "lampa_1_korytarz_1_1_wl"
        tap Program_1.lampa_1_korytarz_1_1_visu
    Lamp1 (390,98 36x36), variable: lampa_1_korytarz_1_1_rel, style: Lamp-Lamp1-Yellow
    Button (23,16 150x30), "lampa_1_pokoj_1_1_wl"
        tap Program_1.lampa_1_pokoj_1_1_visu
    Lamp1 (179,16 36x36), variable: lampa_1_pokoj_1_1_rel, style: Lamp-Lamp1-Yellow
    Button (23,57 150x30), "lampa_1_pokoj_2_1_wl"
        tap Program_1.lampa_1_pokoj_2_1_visu
    Lamp1 (179,52 36x36), variable: lampa_1_pokoj_2_1_rel, style: Lamp-Lamp1-Yellow
    Button (23,101 150x30), "kinkiet_1_pokoj_2_1_wl"
        tap Program_1.kinkiet_1_pokoj_2_1_visu
    Lamp1 (179,100 36x36), variable: kinkiet_1_pokoj_2_1_rel, style: Lamp-Lamp1-Yellow
    Button (233,16 150x30), "lampa_2_korytarz_1_1_wl"
        tap Program_1.lampa_2_korytarz_1_1_VISU
    Lamp1 (390,16 36x36), variable: lampa_2_korytarz_1_1_rel, style: Lamp-Lamp1-Yellow
    Button (233,173 150x30), "lampa_pom_tech_1_1_wl"
        tap Program_1.lampa_pom_tech_1_1_visu
    Lamp1 (390,169 36x36), variable: lampa_pom_tech_1_1_rel, style: Lamp-Lamp1-Yellow
    Button (23,174 150x30), "lampa_1_lazienka_1_1_wl"
        tap Program_1.lampa_1_lazienka_1_1_visu
    Lamp1 (179,170 36x36), variable: lampa_1_lazienka_1_1_rel, style: Lamp-Lamp1-Yellow
    Button (800,597 150x30), "lampa_zew_1_1_wl"
        tap Program_1.lampa_zew_1_1_visu
    Lamp1 (970,596 36x36), variable: lampa_zew_1_1_rel, style: Lamp-Lamp1-Yellow
    Button (796,641 150x30), "lampa_zew_2_1_wl"
        tap Program_1.lampa_zew_2_1_visu
    Lamp1 (966,640 36x36), variable: lampa_zew_2_1_rel, style: Lamp-Lamp1-Yellow
    Button (794,685 150x30), "lampa_zew_3_1_wl"
        tap Program_1.lampa_zew_3_1_visu
    Lamp1 (964,684 36x36), variable: lampa_zew_3_1_rel, style: Lamp-Lamp1-Yellow
    Button (799,727 150x30), "lampa_zew_4_1_wl"
        tap Program_1.lampa_zew_4_1_visu
    Lamp1 (968,723 36x36), variable: lampa_zew_4_1_rel, style: Lamp-Lamp1-Yellow
    Button (492,448 150x30), "lampa_1_pokoj_3_1_wl"
        tap Program_1.lampa_1_pokoj_3_1_visu
    Lamp1 (661,444 36x36), variable: lampa_1_pokoj_3_1_rel, style: Lamp-Lamp1-Yellow
    Button (497,490 141x30), "lampa_1_pom_gosp_1_1_wl"
        tap Program_1.lampa_1_pom_gosp_1_1_visu
    Lamp1 (659,482 36x36), variable: lampa_1_pom_gosp_1_1_rel, style: Lamp-Lamp1-Yellow
    Button (493,534 150x30), "lampa_1_pokoj_4_1_wl"
        tap Program_1.lampa_1_pokoj_4_1_visu
    Lamp1 (662,530 36x36), variable: lampa_1_pokoj_4_1_rel, style: Lamp-Lamp1-Yellow
    Button (491,578 145x28), "lampa_2_pokoj_4_1_wl"
        tap Program_1.lampa_2_pokoj_4_1_visu
    Lamp1 (660,574 36x36), variable: lampa_2_pokoj_4_1_rel, style: Lamp-Lamp1-Yellow
    Button (496,620 150x30), "lampa_1_pokoj_5_1_wl"
        tap Program_1.lampa_1_pokoj_5_1_visu
    Lamp1 (665,616 36x36), variable: lampa_1_pokoj_5_1_rel, style: Lamp-Lamp1-Yellow
    Button (670,30 150x30), "lampa_1_korytarz_2_1_wl"
        tap Program_1.lampa_1_korytarz_2_1_visu
    Lamp1 (839,26 36x36), variable: lampa_1_korytarz_2_1_rel, style: Lamp-Lamp1-Yellow
    Button (666,74 150x30), "led_1_korytarz_2_1_wl"
        tap Program_1.led_1_korytarz_2_1_visu
    Lamp1 (835,70 36x36), variable: led_1_korytarz_2_1_rel, style: Lamp-Lamp1-Yellow
    Button (664,118 150x30), "lampa_1_lazienka_2_1_wl"
        tap Program_1.lampa_1_lazienka_2_1_visu
    Lamp1 (833,114 36x36), variable: lampa_1_lazienka_2_1_rel, style: Lamp-Lamp1-Yellow
    Button (669,160 150x30), "kinkiet_1_lazienka_2_1_wl"
        tap Program_1.kinkiet_1_lazienka_2_1_visu
    Lamp1 (838,156 36x36), variable: kinkiet_1_lazienka_2_1_rel, style: Lamp-Lamp1-Yellow
    Button (663,202 150x30), "kinkiet_2_lazienka_2_1_wl"
        tap Program_1.kinkiet_2_lazienka_2_1_visu
    Lamp1 (832,198 36x36), variable: kinkiet_2_lazienka_2_1_rel, style: Lamp-Lamp1-Yellow
    Button (668,244 150x30), "lampa_1_pralnia_1_1_wl"
        tap Program_1.lampa_1_pralnia_1_1_visu
    Lamp1 (837,240 36x36), variable: lampa_1_pralnia_1_1_rel, style: Lamp-Lamp1-Yellow
    Button (664,288 150x30), "lampa_1_garderoba_1_1_wl"
        tap Program_1.lampa_1_garderoba_1_1_visu
    Lamp1 (833,284 36x36), variable: lampa_1_garderoba_1_1_rel, style: Lamp-Lamp1-Yellow
    Button (662,332 150x30), "os_ogrodu_1_1_wl"
        tap Program_1.os_ogrodu_1_1_visu
    Lamp1 (831,328 36x36), variable: os_ogrodu_1_1_rel, style: Lamp-Lamp1-Yellow
    Button (22,443 150x30), "kinkiet_4_salon_1_1_wl"
        tap Program_1.kinkiet_4_salon_1_1_visu
    Lamp1 (180,440 36x36), variable: kinkiet_4_salon_1_1_rel, style: Lamp-Lamp1-Yellow
    Button (23,217 148x28), "kinkiet_1_lazienka_1_1_wl"
        tap Program_1.kinkiet_1_lazienka_1_1_visu
    Lamp1 (179,213 36x36), variable: kinkiet_1_lazienka_1_1_rel, style: Lamp-Lamp1-Yellow
    Button (495,658 147x26), "kinkiet_1_pokoj_5_1_wl"
        tap Program_1.kinkiet_1_pokoj_5_1_visu
    Lamp1 (664,654 36x36), variable: kinkiet_1_pokoj_5_1_rel, style: Lamp-Lamp1-Yellow
    Button (666,412 150x30), "kinkiet_2_schody_1_1_wl"
        tap Program_1.kinkiet_2_schody_1_1_visu
    Lamp1 (835,408 36x36), variable: kinkiet_2_schody_1_1_rel, style: Lamp-Lamp1-Yellow
    Button (805,521 150x30), "lampa_zew_5_1_wl"
        tap Program_1.lampa_zew_5_1_visu
    Lamp1 (973,513 36x47), variable: lampa_zew_5_1_rel, style: Lamp-Lamp1-Yellow
    Button (276,481 150x30), "Rzut VISU"
        OnMouseUp:  Assign=Visualization_1, Type=Assignment
END_VISUALIZATION

// MyController/Application/Visualization_1
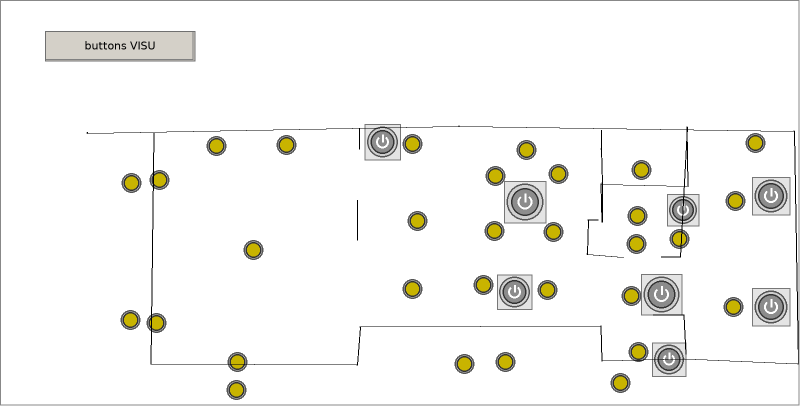
VISUALIZATION Visualization_1  // 800x406
    Lamp1 (630,156 23x28), style: Lamp-Lamp1-Yellow
    Lamp1 (744,129 23x28), style: Lamp-Lamp1-Yellow
    Lamp1 (724,187 23x28), variable: lampa_1_pokoj_2_1_rel, style: Lamp-Lamp1-Yellow
    Lamp1 (722,293 23x28), variable: lampa_1_pokoj_1_1_rel, style: Lamp-Lamp1-Yellow
    Lamp1 (627,338 23x28), variable: lampa_1_przedsionek_1_1_rel, style: Lamp-Lamp1-Yellow
    Lamp1 (609,369 23x28), style: Lamp-Lamp1-Yellow
    Lamp1 (453,350 23x28), style: Lamp-Lamp1-Yellow
    Lamp1 (494,348 23x28), style: Lamp-Lamp1-Yellow
    Lamp1 (484,162 23x28), variable: lampa_1_kuchania_1_1_rel, style: Lamp-Lamp1-Yellow
    Lamp1 (547,160 23x28), variable: lampa_1_kuchania_1_1_rel, style: Lamp-Lamp1-Yellow
    Lamp1 (483,217 23x28), variable: lampa_1_kuchania_1_1_rel, style: Lamp-Lamp1-Yellow
    Lamp1 (542,218 23x28), variable: lampa_1_kuchania_1_1_rel, style: Lamp-Lamp1-Yellow
    Lamp1 (620,282 23x28), variable: lampa_1_korytarz_1_1_rel, style: Lamp-Lamp1-Yellow
    Lamp1 (625,230 23x28), style: Lamp-Lamp1-Yellow
    Lamp1 (626,202 23x28), style: Lamp-Lamp1-Yellow
    Lamp1 (668,225 23x28), variable: kinkiet_1_lazienka_1_1_rel, style: Lamp-Lamp1-Yellow
    Lamp1 (536,276 23x28), variable: lampa_2_korytarz_1_1_rel, style: Lamp-Lamp1-Yellow
    Lamp1 (472,271 23x28), variable: lampa_2_korytarz_1_1_rel, style: Lamp-Lamp1-Yellow
    Lamp1 (401,275 23x28), variable: lampa_2_korytarz_1_1_rel, style: Lamp-Lamp1-Yellow
    Lamp1 (401,130 23x28), variable: kinkiet_1_jadalnia_1_1_rel, style: Lamp-Lamp1-Yellow
    Lamp1 (406,207 23x28), style: Lamp-Lamp1-Yellow
    Lamp1 (226,348 23x28), style: Lamp-Lamp1-Yellow
    Lamp1 (225,376 23x28), style: Lamp-Lamp1-Yellow
    Lamp1 (275,131 23x28), style: Lamp-Lamp1-Yellow
    Lamp1 (205,132 23x28), style: Lamp-Lamp1-Yellow
    Lamp1 (148,166 23x28), style: Lamp-Lamp1-Yellow
    Lamp1 (145,309 23x28), style: Lamp-Lamp1-Yellow
    Lamp1 (120,169 23x28), style: Lamp-Lamp1-Yellow
    Lamp1 (119,306 23x28), style: Lamp-Lamp1-Yellow
    Lamp1 (242,236 23x28), style: Lamp-Lamp1-Yellow
    Lamp1 (515,136 23x28), style: Lamp-Lamp1-Yellow
    Button (45,31 150x30), "buttons VISU"
        OnMouseUp:  Assign=Visualization, Type=Assignment
    PowerSwitch (504,180 42x44), variable: Program_1.lampa_1_kuchania_visu, behaviour: TAP, style: Switch-PowerSwitch-Gray
    PowerSwitch (665,194 36x32), variable: Program_1.kinkiet_1_lazienka_1_1_visu, behaviour: TOGGLE, style: Switch-PowerSwitch-Gray
    PowerSwitch (641,273 41x43), variable: Program_1.lampa_1_korytarz_1_1_visu, behaviour: TAP, style: Switch-PowerSwitch-Gray
    PowerSwitch (497,271 35x42), variable: Program_1.lampa_2_korytarz_1_1_VISU, behaviour: TAP, style: Switch-PowerSwitch-Gray
    PowerSwitch (652,335 34x49), variable: Program_1.lampa_1_przedsionek_1_1_visu, behaviour: TAP, style: Switch-PowerSwitch-Gray
    PowerSwitch (364,124 37x36), variable: Program_1.kinkiet_1_jadalnia_1_1_visu, behaviour: TAP, style: Switch-PowerSwitch-Gray
    PowerSwitch (748,288 46x38), variable: Program_1.lampa_1_pokoj_1_1_visu, behaviour: TAP, style: Switch-PowerSwitch-Gray
    PowerSwitch (748,177 46x38), variable: Program_1.lampa_1_pokoj_2_1_visu, behaviour: TAP, style: Switch-PowerSwitch-Gray
    Polyline (87,132) (87,133) (459,126) (794,131) (798,364) (684,359) (602,361) (601,326) (360,327) (357,365) (151,364) (154,133)
    Polyline (601,130) (601,149) (602,183) (602,222) (601,184) (688,186) (687,127) (680,257) (661,257)
    Polyline (598,220) (588,220) (587,254) (623,257)
    Polyline (686,354) (684,315) (653,315)
    Polyline (359,128) (359,149)
    Polyline (357,200) (357,240)
END_VISUALIZATION
